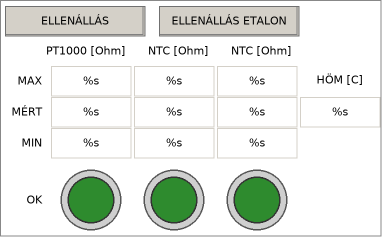
VISUALIZATION Vegmero_ellenallas  // 382x237
    Lamp1 (56,165 70x70), variable: NOT VEGMERO.bPTRES_OK, style: Lamp-Lamp1-Red
    Lamp1 (139,165 70x70), variable: NOT VEGMERO.bNTCRES_OK, style: Lamp-Lamp1-Red
    Button (5,6 140x30), "ELLENÁLLÁS", input disabled if: VEGMERO.s_InCommand<>''
        OnMouseUp: execute { VEGMERO.s_InCommand:='ELLENALLAS'; }
    Textfield (51,97 80x30), "%s", text variable: VEGMERO.rPTRES
    Textfield (134,97 80x30), "%s", text variable: VEGMERO.rNTCRES
    Textfield (51,128 80x30), "%s", text variable: VEGMERO.PTRES_MIN
    Textfield (51,66 80x30), "%s", text variable: VEGMERO.PTRES_MAX
    Textfield (134,128 80x30), "%s", text variable: VEGMERO.NTCRES_MIN
    Textfield (134,66 80x30), "%s", text variable: VEGMERO.NTCRES_MAX
    Textfield (300,97 80x30), "%s", text variable: VEGMERO.rTemp
    Label (5,102 40x20), "MÉRT"
    Label (41,41 90x20), "PT1000 [Ohm]"
    Label (143,41 71x20), "NTC [Ohm]"
    Label (305,70 70x20), "HÖM [C]"
    Button (159,6 140x30), "ELLENÁLLÁS ETALON", input disabled if: VEGMERO.s_InCommand<>''
        OnMouseUp: execute { VEGMERO.s_InCommand:='ELLENALLASETALON'; }
    Label (5,71 40x20), "MAX"
    Label (5,133 40x20), "MIN"
    Label (5,190 40x20), "OK"
    Lamp1 (56,165 70x70), variable: VEGMERO.bPTRES_OK, invisible if: NOT VEGMERO.bPTRES_OK AND VEGMERO.bPTRES_MERVE, style: Lamp-Lamp1-Green
    Lamp1 (139,165 70x70), variable: VEGMERO.bNTCRES_OK, invisible if: NOT VEGMERO.bNTCRES_OK AND VEGMERO.bNTCRES_MERVE, style: Lamp-Lamp1-Green
    Label (226,41 71x20), "NTC [Ohm]"
    Textfield (217,97 80x30), "%s", text variable: VEGMERO.rNTCRES2
    Textfield (217,128 80x30), "%s", text variable: VEGMERO.NTCRES2_MIN
    Textfield (217,66 80x30), "%s", text variable: VEGMERO.NTCRES2_MAX
    Lamp1 (222,165 70x70), variable: NOT VEGMERO.bNTCRES2_OK, style: Lamp-Lamp1-Red
    Lamp1 (222,165 70x70), variable: VEGMERO.bNTCRES2_OK, invisible if: NOT VEGMERO.bNTCRES2_OK AND VEGMERO.bNTCRES2_MERVE, style: Lamp-Lamp1-Green
END_VISUALIZATION

(* stored: Version 1.1.0.1, ProductVersion 3.1.4024.11
   Visu Vegmero_ellenallas: Id {0aee45cc-3cc2-481e-a5df-d47743b5340b} *)
